{attribute 'GeneratedUsingTerminal: EL3773-0000-0018'}
{attribute addProperty BoxType "EL3773-0000-0018"}
{attribute addProperty Id "I1_SamplesAT %I*I1_Samples_2D13B74B20"}
{attribute addProperty CRC "1292205132"}
{attribute addProperty Size "20"}
TYPE L1_Current_Samples_4D057C4C :
STRUCT
	{attribute addProperty Name "I1_Samples"}
	I1_Samples AT %I* : I1_Samples_2D13B74B;
END_STRUCT
END_TYPE

(* stored: Version 1.2.0.0, ProductVersion 3.1.4024.9
   DUT L1_Current_Samples_4D057C4C: Id {2d46559f-6560-46a3-ace1-cf042e0e7b4a} *)
